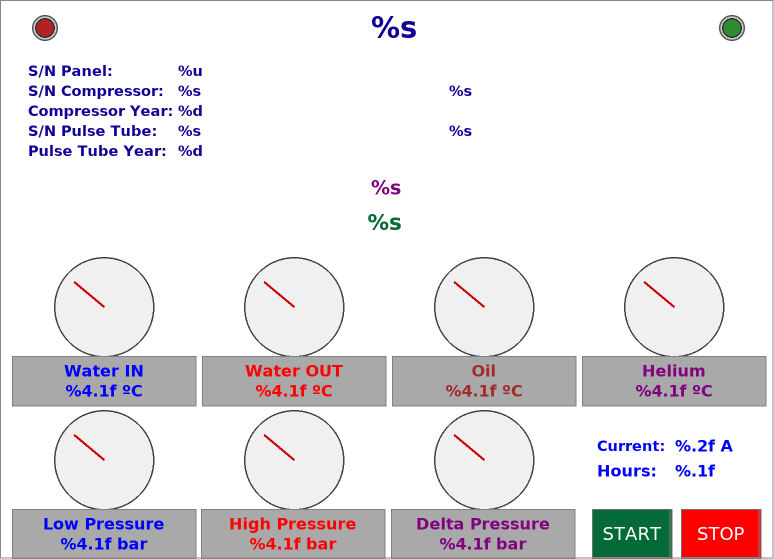
VISUALIZATION GUI_TEMPLATE_CRYO_CPA  // 774x559
VAR_IN_OUT
	m_Instance:	FB_CRYO_CPA;
END_VAR
    Rectangle (80,10 629x35), "%s", text variable: m_Instance.stat.sModelNumber
    Rectangle (10,207 750x30), "%s", text variable: m_Instance.stat.sError, invisible if: (m_Instance.stat.nStatusCode<>2)
    Meter180 (4,410 200x100), value: m_Instance.stat.lrLowPressure, style: Meter-Meter180-Gray, scale format: %.0f, scale 0..30
    Rectangle (12,509 184x50), "Low Pressure %4.1f bar", text variable: m_Instance.stat.lrLowPressure
    Meter180 (194,410 200x100), value: m_Instance.stat.lrHighPressure, style: Meter-Meter180-Gray, scale format: %.0f, scale 0..30
    Rectangle (201,509 184x50), "High Pressure %4.1f bar", text variable: m_Instance.stat.lrHighPressure
    Lamp1 (717,13 30x30), tooltip "If ON, compressor is running", variable: m_Instance.stat.bSystemOn, style: Lamp-Lamp1-Green
    Rectangle (10,208 750x30), "%s", text variable: m_Instance.stat.sAlarm, invisible if: (m_Instance.stat.nStatusCode<>1)
    Rectangle (231,206 308x33), "%s", text variable: m_Instance.stat.sStatusOK, invisible if: (m_Instance.stat.nStatusCode<>0 or m_Instance.stat.nOperatingState <>3)
    Meter180 (4,257 200x100), value: m_Instance.stat.lrCoolantInTemp, style: Meter-Meter180-Gray, scale format: %.0f, scale 0..60
    Rectangle (12,356 184x50), "Water IN %4.1f ºC", text variable: m_Instance.stat.lrCoolantInTemp
    Meter180 (194,257 200x100), value: m_Instance.stat.lrCoolantOutTemp, style: Meter-Meter180-Gray, scale format: %.0f, scale 0..60
    Rectangle (202,356 184x50), "Water OUT %4.1f ºC", text variable: m_Instance.stat.lrCoolantOutTemp
    Meter180 (384,257 200x100), value: m_Instance.stat.lrOilTemp, style: Meter-Meter180-Gray, scale format: %.0f, scale 0..60
    Rectangle (392,356 184x50), "Oil %4.1f ºC", text variable: m_Instance.stat.lrOilTemp
    Meter180 (574,257 200x100), value: m_Instance.stat.lrHeliumTemp, style: Meter-Meter180-Gray, scale format: %.0f, scale 0..100
    Rectangle (582,356 184x50), "Helium %4.1f ºC", text variable: m_Instance.stat.lrHeliumTemp
    Rectangle (672,431 95x30), "%.2f A", text variable: m_Instance.stat.lrMotorCurrent
    Rectangle (672,456 95x30), "%.1f", text variable: m_Instance.stat.lrHoursOfOperation
    Rectangle (140,173 493x30), "%s", tooltip "Operational State", text variable: m_Instance.stat.sOperatingState
    Rectangle (175,60 231x22), "%u", text variable: m_Instance.stat.nPanelSerialNumber
    Rectangle (175,80 270x22), "%s", text variable: m_Instance.in_sSN_Compressor
    Rectangle (175,120 270x22), "%s", text variable: m_Instance.in_sSN_PulseTube
    Label (25,60 145x22), "S/N Panel:"
    Label (25,80 145x22), "S/N Compressor:"
    Label (25,120 145x22), "S/N Pulse Tube:"
    Rectangle (594,431 75x30), "Current:"
    Rectangle (594,456 75x30), "Hours:"
    Meter180 (384,410 200x100), value: m_Instance.stat.lrDeltaPressureAverage, style: Meter-Meter180-Gray, scale format: %.0f, scale 0..30
    Rectangle (391,509 184x50), "Delta Pressure %4.1f bar", text variable: m_Instance.stat.lrDeltaPressureAverage
    Label (25,140 145x22), "Pulse Tube Year:"
    Rectangle (175,140 90x22), "%d", text variable: m_Instance.in_nYear_PulseTube
    Label (25,100 145x22), "Compressor Year:"
    Rectangle (175,100 90x22), "%d", text variable: m_Instance.in_nYear_Compressor
    Rectangle (446,80 270x22), "%s", text variable: m_Instance.stat.sServiceDue_Compressor, invisible if: m_Instance.stat.bServiceDue_Compressor=FALSE
        p55702900: m_Instance.stat.wColour_Compressor
    Rectangle (446,120 270x22), "%s", text variable: m_Instance.stat.sServiceDue_PulseTube, invisible if: m_Instance.stat.bServiceDue_PulseTube=FALSE
        p55702900: m_Instance.stat.wColour_PulseTube
    Button (592,509 80x50), "START", input disabled if: m_Instance.stat.bSystemOn
        OnMouseClick: execute { m_Instance.ctrl.nDevCommand := E_CRYO_CPA_CMDS.START; m_Instance.ctrl.bExecute := TRUE; }
    Button (681,509 80x50), "STOP", input disabled if: NOT m_Instance.stat.bSystemOn
        OnMouseClick: execute { m_Instance.ctrl.nDevCommand := E_CRYO_CPA_CMDS.STOP; m_Instance.ctrl.bExecute := TRUE; }
    Lamp1 (30,13 30x30), tooltip "If ON, compressor is simulated", variable: m_Instance.stat.bSimulation, invisible if: m_Instance.stat.bSimulation=false, style: Lamp-Lamp1-Red
END_VISUALIZATION

(* stored: Version 1.1.0.1, ProductVersion 3.1.4024.9
   Visu GUI_TEMPLATE_CRYO_CPA: Id {d996caad-054e-47b3-a9f8-f22c6178eb5e} *)
